Staubli VAL3: calculate_rc.pgx

program calculate_rc(num x_nNum_index, num x_nNum_choose, num& x_nNum_cRow, num& x_nNum_cCol)
  local num l_nNum_lCol
  local num l_nNum_lRow
begin

  call return_config(x_nNum_choose,l_nNum_lRow,l_nNum_lCol)

  //Quotien
  x_nNum_cRow = roundDown(x_nNum_index / (l_nNum_lCol + 1))
  //Modulo reminder
  x_nNum_cCol = x_nNum_index % (l_nNum_lCol+1)


end
